PROGRAM MAIN
VAR
END_VAR

ST_MotionControl();
ST_Kapsekvens();
ST_Homing();
LD_Spantransportor();

END_PROGRAM

(* stored: Version 1.1.0.1, ProductVersion 3.1.4024.10
   POU MAIN: Id {64bf3122-88c5-4b02-8950-c8e656632d3c}, SpecialFunc None *)
